FUNCTION_BLOCK Axis
//VAR_INPUT	
//END_VAR
VAR_OUTPUT
	Axis_Error			: BOOL;				// Error signal
	Axis_ErrorID		: UDINT;			// Error ID
	Axis_Moves			: BOOL;				// Status of moving
END_VAR
VAR
	// =============== Done signals MC Block =================
	JogDone			    : BOOL;					// Status of function block MC_Jog
	ResetDone		    : BOOL;					// Status of function block MC_Reset
	HaltDone		    : BOOL;					// Status of function block MC_Halt
	HomeDone		    : BOOL;					// Status of function block MC_Home
  MoveAbsoluteDone : BOOL;        // Status of function block MC_MoveAbsolute
  ExtSetPiontDone 	: BOOL;         		// Status of function block MC_ExtSetPointGenDisable

	// =============== Control variables ======================
	//Home_Back_Start	: BOOL;
	//Drive_Home		: BOOL;
	
	// =============== State variables ========================
	Power_StatusEnable	: BOOL;					// Enable feedback
	
	// =============== Velocity, override =====================
	Velocity_Jog		: LREAL;				// Jog velocity
	Velocity_Move		: LREAL;				// Target velocity
	Velocity_Home		: LREAL;				// Home1 velocity
  Velocity_Home2    : LREAL;        // Home1 velocity   
	Velocity_Absolute	: LREAL;				// MoveAbsolute velocity
	Velocity_Relative	: LREAL;				// MoveRelative velocity
	fOverride 			: LREAL := 100.0;		// Override 100%
	
	// =============== Trigger function blocks ================
	
	TriggerHalt	: R_TRIG;				// Trigger to recognize rising edge of halt input
	TriggerReset : R_TRIG;				// Trigger to recognize rising edge of reset input
	
	// =============== Axis reference =========================
	AxisRef			: AXIS_REF;				// Axis reference (process data plc/nc)
	
	// =============== About axis turque ====================
	Axis_Current_Turque 	: INT;
  	Axis_Max_Turque       	: INT;
	// ================= Sensor FeedBack ====================
  Proximity_Switch      : DINT;
  
	// =============== Motion function blocks =================
	Axis_Power 			: MC_Power;				// FB for enable and override			[上电]
	Axis_Home			: MC_Home;				// FB for axis home						[找零]
	Axis_Reset 			: MC_Reset;				// FB to reset axis						[复位]
	Axis_Jog			: MC_Jog;				// FB to jog axis						[点动]
	Axis_Stop 			: MC_Stop;				// FB to stop axis						[停止]
	Axis_Halt			: MC_Halt;				// FB to halt axis						[停止]
	Axis_Move			: MC_MoveVelocity;		// FB to move axis (velocity movement)	[匀速运动]
	Axis_MoveAbsolute 	: MC_MoveAbsolute;		// FB to move axis absolutely			[绝对位置运动]
	Axis_MoveRelative	: MC_MoveRelative;		// FB to move axis relatively			[相对位置运动]
  	Axis_ActPosition  : MC_ReadActualPosition; // FB to read the actual position of axis  [读取电机轴的实际位置]
	Axis_Delay			: Delay;				// FB to operate the delay program		[延迟程序]
	Axis_ExtSetPiontEnable	: MC_ExtSetPointGenEnable;	// FB to enable extsetpoint		[外部函数发生使能]
	Axis_ExtSetPiontDisable	: MC_ExtSetPointGenDisable;	// FB to disable extsetpoint	[外部函数结束使能]
  
  // =============== Timer =================
  Delay         : TON;          //[定时器]
END_VAR

PROPERTY ActPosition : LREAL
GET
Axis_ActPosition( Axis:= AxisRef, Enable:= TRUE );
ActPosition := Axis_ActPosition.Position;
END_GET
END_PROPERTY

PROPERTY Current_Turque_Value : INT
GET
Current_Turque_Value := Axis_Current_Turque;
END_GET
SET
Axis_Current_Turque := Current_Turque_Value;
END_SET
END_PROPERTY

METHOD ExtSetPoint
VAR_INPUT
	Drive_ExtSetPointEnable 	: BOOL;		// 使能外部信号开始信号
	Drive_ExtSetPointDisable 	: BOOL;		// 使能外部信号结束信号
	ExSetPosition				: LREAL;	// 外部信号位置
	//Axis_Current_Turque 		: INT;		// 边界条件：丝杠位置到达两端卡死
END_VAR
// =======================外部信号发生程序==========================

IF NOT Axis_ExtSetPiontEnable.Error THEN
	Axis_ExtSetPiontEnable(	Axis:= AxisRef, 
							Execute:= Drive_ExtSetPointEnable, 
							Position:= ExSetPosition, 
							PositionType:= POSITIONTYPE_ABSOLUTE );
END_IF

IF Axis_ExtSetPiontEnable.Done THEN
	ExtSetPiontDone := 1;
	MC_ExtSetPointGenFeed(	Position:= ExSetPosition, 
							Velocity:= 10, 
							Acceleration:= 10, 
							Direction:= 1, 		// 1 = positive direction
							Axis:= AxisRef );
END_IF	

IF NOT Axis_ExtSetPiontDisable.Error THEN 
	Axis_ExtSetPiontDisable(	Axis:= AxisRef, 
								Execute:= Drive_ExtSetPointDisable);
END_IF
								
IF Axis_ExtSetPiontEnable.Error OR Axis_ExtSetPiontDisable.Error OR ABS(Axis_Current_Turque) > Axis_Max_Turque THEN
	IF Axis_ExtSetPiontEnable.Error OR Axis_ExtSetPiontDisable.Error THEN
		Axis_Error		:= TRUE;
		Axis_ErrorID 	:= Axis_Home.ErrorID;
	END_IF
	Axis_ExtSetPiontEnable(	Axis:= AxisRef, 
							Execute:= 0 );
	Axis_ExtSetPiontDisable(	Axis:= AxisRef, 
								Execute:= 1);
END_IF
END_METHOD

METHOD Halt : BOOL
VAR_INPUT
	DriveHalt		: BOOL;					// Request stop
END_VAR
// =======================电机运动停止程序==========================

IF DriveHalt THEN
	// Move Execute FALSE
	Axis_Move(	Execute	:= FALSE,
				Axis 	:= AxisRef);
ELSE
	// Reset done signal
	HaltDone := FALSE;
END_IF

// Trigger
TriggerHalt(CLK := DriveHalt);

IF TriggerHalt.Q THEN
	Axis_Halt(	Execute	:= TRUE,
				Axis 	:= AxisRef);
ELSE
	Axis_Halt(Axis := AxisRef);
END_IF

// Done / Error / Command aborted
IF Axis_Halt.Done OR Axis_Halt.Error OR Axis_Halt.CommandAborted THEN
	Axis_Error		:= Axis_Halt.Error;
	Axis_ErrorID 	:= Axis_Halt.ErrorID;
	HaltDone 		:= Axis_Halt.Done;
	
	Axis_Move(	Execute	:= FALSE,
				Axis 	:= AxisRef);
				
	Axis_Halt(	Execute	:= FALSE,
				Axis 	:= AxisRef);
END_IF

// =========================================================
END_METHOD

METHOD Home
VAR_INPUT
	//Back_Start 				: BOOL;
	//Velocity_Home	:LREAL;
	//Axis_Current_Turque 	: INT;
	Drive_Home				: BOOL;
END_VAR

VAR
	HomeSet					: BOOL;
END_VAR
// =======================找零程序==========================
// 找零程序过程为：先让丝杠回退，到达机械限位后停止,并用程序将该位置置为零位

//======================丝杠回退========================
Jog_Backward(Drive_Jog_Backward:= Drive_Home);
Jog_Velocity := Velocity_Home;
	
IF NOT Axis_Home.Error THEN
	IF ABS(Axis_Current_Turque) > Axis_Max_Turque AND NOT HomeDone THEN
		Drive_Home :=0;
		Jog_Backward(Drive_Jog_Backward:= Drive_Home);
		Delay(IN:= NOT Delay.Q, PT:=T#200MS, Q=> , ET=> );
		Axis_Home( 	Axis:= AxisRef, 
					Execute:= Delay.Q, 
					Position:= 0, 
					HomingMode:= MC_Direct);
		HomeDone := Axis_Home.Done;
	END_IF
	IF HomeDone THEN
		Move_Absolute(Drive_Move_Absolute:= TRUE, Absolute_Position:= 10 );
		IF Axis_MoveAbsolute.Done THEN
			HomeDone := FALSE;
		END_IF
	END_IF
END_IF

(*IF HomeSet THEN
	Jog_Backward(Drive_Jog_Backward:= 0,  Axis_Current_Turque:= Axis_Current_Turque);
	HomeDone := 1;
END_IF*)

IF Axis_Home.Error OR Axis_Home.CommandAborted OR ABS(Axis_Current_Turque) < Axis_Max_Turque THEN
	IF Axis_Jog.Error THEN
		Axis_Error		:= TRUE;
		Axis_ErrorID 	:= Axis_Home.ErrorID;
	END_IF
	Axis_Home( 	Axis:= AxisRef, 
				Execute:= FALSE);
END_IF

// =========================================================
END_METHOD

PROPERTY Home_Velocity : LREAL
GET
Home_Velocity := Velocity_Home;
END_GET
SET
Velocity_Home := Home_Velocity;
END_SET
END_PROPERTY

METHOD Home2 : BOOL
VAR_INPUT
	Drive_Home		: BOOL;
END_VAR
// =======================找零程序==========================
// 找零程序过程为：先让丝杠回退，当传感器检测到金属表面并反馈信号后, 程序将该位置置为零位

//======================丝杠回退========================
Jog_Backward(Drive_Jog_Backward:= Drive_Home);
Jog_Velocity := Velocity_Home2;
	
IF NOT Axis_Home.Error THEN
	IF ABS(Proximity_Switch) = 64028672 AND NOT HomeDone THEN
		Drive_Home :=0;
		Jog_Backward(Drive_Jog_Backward:= Drive_Home);
		Delay(IN:= NOT Delay.Q, PT:=T#200MS, Q=> , ET=> );
		Axis_Home( 	Axis:= AxisRef, 
					Execute:= Delay.Q,
					Position:= 0, 
					HomingMode:= MC_Direct);
		HomeDone := Axis_Home.Done;
	END_IF
	IF HomeDone THEN
		Move_Absolute(Drive_Move_Absolute:= TRUE, Absolute_Position:= 20);
		IF Axis_MoveAbsolute.Done THEN
			HomeDone := FALSE;
		END_IF
	END_IF
END_IF

(*IF HomeSet THEN
	Jog_Backward(Drive_Jog_Backward:= 0,  Axis_Current_Turque:= Axis_Current_Turque);
	HomeDone := 1;
END_IF*)

IF Axis_Home.Error OR Axis_Home.CommandAborted OR ABS(Axis_Current_Turque) < Axis_Max_Turque THEN
	IF Axis_Jog.Error THEN
		Axis_Error		:= TRUE;
		Axis_ErrorID 	:= Axis_Home.ErrorID;
	END_IF
	Axis_Home( 	Axis:= AxisRef, 
				Execute:= FALSE);
END_IF

// =========================================================
END_METHOD

PROPERTY Home2_Velocity : LREAL
GET
Home2_Velocity := Velocity_Home2;
END_GET
SET
Velocity_Home2 := Home2_Velocity;
END_SET
END_PROPERTY

METHOD Jog_Backward
VAR_INPUT
	Drive_Jog_Backward	: BOOL;				//点动后退使能信号
	//Velocity_Jog		: LREAL;			//点动速度
	//Axis_Current_Turque : INT;				//边界条件：丝杠位置到达两端卡死
END_VAR
// =======================点动后退==========================
// 点动后退用在找零中的位置移动

IF NOT Axis_Jog.Error THEN
	Axis_Jog( 	Axis:= AxisRef, 
				JogForward:= 0, 
				JogBackwards:= Drive_Jog_Backward, 
				Mode:= MC_JOGMODE_CONTINOUS, 
				Velocity:= Velocity_Jog);
END_IF

IF Axis_Jog.Error OR Axis_Jog.CommandAborted OR ABS(Axis_Current_Turque) > Axis_Max_Turque THEN
	IF Axis_Jog.Error THEN
		Axis_Error		:= TRUE;
		Axis_ErrorID 	:= Axis_Jog.ErrorID;
	END_IF
	
	Axis_Jog(	JogForward:= 0, 
				JogBackwards:= 0, 
				Axis := AxisRef);
END_IF

(*IF ABS(Axis_Current_Turque) <1000 AND JogDone =1 THEN
	Axis_Jog(	JogForward:= 0, 
				JogBackwards:= 0, 
				Axis := AxisRef);
	JogDone :=0;
END_IF*)
				
// =========================================================
END_METHOD

METHOD Jog_Forward : BOOL
VAR_INPUT
	Drive_Jog_Forward	: BOOL;				//点动前进使能信号
	//Velocity_Jog		: LREAL;			//点动速度
	//Axis_Current_Turque : INT;				//边界条件：丝杠位置到达两端卡死
END_VAR
// =======================点动前进==========================


IF NOT Axis_Jog.Error THEN
	Axis_Jog( 	Axis:= AxisRef, 
				JogForward:= Drive_Jog_Forward, 
				JogBackwards:= 0, 
				Mode:= MC_JOGMODE_CONTINOUS, 
				Velocity:= Velocity_Jog);
END_IF

IF Axis_Jog.Error OR Axis_Jog.CommandAborted OR ABS(Axis_Current_Turque) > Axis_Max_Turque THEN
	IF Axis_Jog.Error THEN
		Axis_Error		:= TRUE;
		Axis_ErrorID 	:= Axis_Jog.ErrorID;
	END_IF
	
	Axis_Jog(	JogForward:= 0, 
				JogBackwards:= 0, 
				Axis := AxisRef);
END_IF

(*IF ABS(Axis_Current_Turque) <1000 AND JogDone =1 THEN
	Axis_Jog(	JogForward:= 0, 
				JogBackwards:= 0, 
				Axis := AxisRef);
	JogDone :=0;
END_IF*)
				
// =========================================================
END_METHOD

// =======================读写点动程序中的速度值==========================

PROPERTY Jog_Velocity : LREAL
GET
Jog_Velocity := Velocity_Jog;
END_GET
SET
Velocity_Jog := Jog_Velocity;
END_SET
END_PROPERTY

PROPERTY Max_Turque_Value : INT
SET
Axis_Max_Turque := Max_Turque_Value;
END_SET
END_PROPERTY

METHOD Move_Absolute
VAR_INPUT
	Drive_Move_Absolute : BOOL;				// 运动使能信号
	Absolute_Position	: LREAL;			// 绝对运动位置
	//Move_Velocity		: LREAL;			// 运动速度
	//Axis_Current_Turque : INT;			// 边界条件：丝杠位置到达两端卡死
END_VAR
// =======================绝对运动==========================

IF NOT Axis_MoveAbsolute.Error THEN
	Axis_MoveAbsolute(	Axis:= AxisRef, 
						Execute:= Drive_Move_Absolute, 
						Position:= Absolute_Position, 
						Velocity:= Velocity_Absolute, 
						BufferMode:= MC_Aborting );
	MoveAbsoluteDone := Axis_MoveAbsolute.Done;			// 运动到指定位置后置位
END_IF

IF Axis_MoveAbsolute.Error OR Axis_MoveAbsolute.CommandAborted OR ABS(Axis_Current_Turque) > Axis_Max_Turque THEN
	IF Axis_MoveAbsolute.Error THEN
		Axis_Error		:= TRUE;
		Axis_ErrorID 	:= Axis_MoveAbsolute.ErrorID;
	END_IF
	
	Axis_MoveAbsolute(	Axis:= AxisRef, 
						Execute:= 0, 
						BufferMode:= MC_Aborting);
END_IF

// =========================================================
END_METHOD

// =======================读写绝对运动程序中的速度值==========================

PROPERTY Move_Absolute_Velocity : LREAL
GET
Move_Absolute_Velocity := Velocity_Absolute;
END_GET
SET
Velocity_Absolute := Move_Absolute_Velocity;
END_SET
END_PROPERTY

METHOD Move_Backward
VAR_INPUT
	Move_Backward_Start : BOOL;					//匀速后退使能信号
	//Axis_Current_Turque : INT;					//边界条件：丝杠位置到达两端卡死
END_VAR
// =======================匀速后退==========================

// Not error
IF NOT Axis_Move.Error THEN
	Axis_Move(	Execute 	:= Move_Backward_Start,
				Velocity 	:= Velocity_Move,
				Direction 	:= MC_Negative_Direction,
				Axis 		:= AxisRef );
END_IF

// Error / Command aborted
IF Axis_Move.Error OR Axis_Move.CommandAborted OR ABS(Axis_Current_Turque) > Axis_Max_Turque THEN
	IF Axis_Move.Error THEN
		Axis_Error		:= TRUE;
		Axis_ErrorID 	:= Axis_Move.ErrorID;
	END_IF
	
	Axis_Move(	Execute	:= FALSE,
				Axis 	:= AxisRef);
END_IF

// =========================================================
END_METHOD

METHOD Move_Fordward
VAR_INPUT
	Move_Forward_Start : BOOL;					//匀速前进使能信号
	//Axis_Current_Turque : INT;					//边界条件：丝杠位置到达两端卡死
END_VAR
// =======================匀速前进==========================

// Not error
IF NOT Axis_Move.Error THEN
	Axis_Move(	Execute 	:= Move_Forward_Start,
				Velocity 	:= Velocity_Move,
				Direction 	:= MC_Positive_Direction,
				Axis 		:= AxisRef );
END_IF

// Error / Command aborted
IF Axis_Move.Error OR Axis_Move.CommandAborted OR ABS(Axis_Current_Turque) > Axis_Max_Turque THEN
	IF Axis_Move.Error THEN
		Axis_Error		:= TRUE;
		Axis_ErrorID 	:= Axis_Move.ErrorID;
	END_IF
	
	Axis_Move(	Execute	:= FALSE,
				Axis 	:= AxisRef);
END_IF

// =========================================================
END_METHOD

METHOD Move_Relative
VAR_INPUT
	Drive_Move_Relative		: BOOL;				// 运动使能信号
	Relative_Position		: LREAL;			// 相对运动位置
	//Move_Velocity			: LREAL;			// 运动速度
	//Axis_Current_Turque 	: INT;				// 边界条件：丝杠位置到达两端卡死
END_VAR
// =======================相对运动==========================

IF NOT Axis_MoveRelative.Error THEN
	Axis_MoveRelative(	Axis:= AxisRef, 
						Execute:= Drive_Move_Relative, 
						Distance:= Relative_Position, 
						Velocity:= Velocity_Relative, 
						BufferMode:= MC_Aborting );
END_IF

IF Axis_MoveRelative.Error OR Axis_MoveRelative.CommandAborted OR ABS(Axis_Current_Turque) > Axis_Max_Turque THEN
	IF Axis_MoveRelative.Error THEN
		Axis_Error		:= TRUE;
		Axis_ErrorID 	:= Axis_MoveRelative.ErrorID;
	END_IF
	
	Axis_MoveRelative(	Axis:= AxisRef, 
						Execute:= 0, 
						BufferMode:= MC_Aborting);
END_IF

// =========================================================
END_METHOD

// =======================读写相对运动程序中的速度值==========================

PROPERTY Move_Relative_Velocity : LREAL
GET
Move_Relative_Velocity := Velocity_Relative;
END_GET
SET
Velocity_Relative := Move_Relative_Velocity;
END_SET
END_PROPERTY

PROPERTY Move_Velocity : LREAL
GET
Move_Velocity := Velocity_Move;
END_GET
SET
Velocity_Move :=Move_Velocity :=10;
END_SET
END_PROPERTY

METHOD Power
VAR_INPUT
	Axis_Enable : BOOL;
END_VAR
// =======================上电程序==========================

Axis_Power(	Enable 			:= Axis_Enable, 
			Enable_Positive	:= Axis_Enable, 
			Enable_Negative	:= Axis_Enable, 
			Override		:= fOverride,
			Axis			:= AxisRef,
			Status			=> Power_StatusEnable);
			
IF Axis_Power.Error THEN
	Axis_Error		:= TRUE;
	Axis_ErrorID 	:= Axis_Power.ErrorID;
END_IF

AxisRef.ReadStatus();

Axis_Moves := AxisRef.Status.Moving;

// ==========================================================
END_METHOD

PROPERTY Proximity_Switch_FeedBack : DINT
SET
Proximity_Switch := Proximity_Switch_FeedBack;
END_SET
END_PROPERTY

METHOD Reset
VAR_INPUT
	Drive_Reset		: BOOL;					// Request reset
END_VAR
// =====================驱动重置程序==========================

IF NOT Drive_Reset THEN
	ResetDone 	:= FALSE;
END_IF

// Trigger(触发器)
TriggerReset(CLK := Drive_Reset);

IF TriggerReset.Q THEN
	HaltDone 	:= FALSE;
	
	Axis_Reset(Execute := TRUE, Axis := AxisRef);
ELSE
	Axis_Reset(Axis := AxisRef);
END_IF

// Done / Error
IF Axis_Reset.Done OR Axis_Reset.Error THEN
	Axis_Error		:= Axis_Reset.Error;
	Axis_ErrorID 	:= Axis_Reset.ErrorID;
	ResetDone 		:= Axis_Reset.Done;

	Axis_Reset(	Execute	:= FALSE, Axis 	:= AxisRef);
END_IF

// =========================================================
END_METHOD

PROPERTY State_ExtSetPiontDone : BOOL
GET
State_ExtSetPiontDone := ExtSetPiontDone;
END_GET
END_PROPERTY

// =======================回零结束信号==========================

PROPERTY State_HomeDone : BOOL
GET
State_HomeDone := HomeDone;
END_GET
END_PROPERTY

// =======================点动结束信号==========================

PROPERTY State_JogDone : BOOL
GET
State_JogDone := JogDone;
END_GET
END_PROPERTY

PROPERTY State_MoveAbsoluteDone : BOOL
GET
State_MoveAbsoluteDone := MoveAbsoluteDone;
END_GET
END_PROPERTY

// =======================上电状态信号==========================

PROPERTY State_PowerStatus : BOOL
GET
State_PowerStatus := Power_StatusEnable;
END_GET
END_PROPERTY

// =======================复位结束信号==========================

PROPERTY State_ResetDone : BOOL
GET
State_ResetDone := ResetDone;
END_GET
END_PROPERTY

END_FUNCTION_BLOCK

(* stored: Version 1.1.0.1, ProductVersion 3.1.4020.12
   POU Axis: Id {752ec826-01be-4872-838e-fdec6a999a4b}, SpecialFunc None
   Property ActPosition: Id {3015e613-88a6-44b7-bfd3-2c06df6f075d}
   Get Get: Id {a1550c61-e344-45b9-84a9-b4c92d3e44f5}
   Property Current_Turque_Value: Id {3a2f771d-3376-4640-bd97-650af6e34455}
   Get Get: Id {cf61b5f8-2ee8-4892-af0b-6df01ee01050}
   Set Set: Id {454d6b57-9848-48a1-bdc6-2e4c4bcfbc97}
   Method ExtSetPoint: Id {e3dd3d6b-d150-49a2-a8d7-a7990a606e4c}
   Method Halt: Id {d7ff254f-2dd7-462f-bdbd-9197c2ffdaa3}
   Method Home: Id {313e1eef-e597-492a-a006-a8453e584cfd}
   Property Home_Velocity: Id {075d0823-6614-4698-9d00-5a9266b58e8c}
   Get Get: Id {337c8281-9e84-4066-80f8-1804a324ddb1}
   Set Set: Id {28f71fe8-0908-4a45-b6fa-862d0622a7a8}
   Method Home2: Id {538e8ca7-d46b-41f9-930c-142666bfb84c}
   Property Home2_Velocity: Id {29542bf1-ba67-49a9-803d-762403c92f58}
   Get Get: Id {fe78f786-10a8-4f98-9e65-95fb7c4427c2}
   Set Set: Id {7e1f886e-1b8d-4d9a-9fc1-c6d7443f0295}
   Method Jog_Backward: Id {99d13956-4937-48a4-92d1-297e5120f462}
   Method Jog_Forward: Id {9deceb4f-22e3-43d3-abba-cc65da0a988f}
   Property Jog_Velocity: Id {fbf70f23-ccbc-42f7-9290-364343308531}
   Get Get: Id {777f885d-c13b-46bb-a81c-11c9d0c034b5}
   Set Set: Id {3493f918-b8b5-4bfd-88eb-49ef90625a72}
   Property Max_Turque_Value: Id {c8624b49-e9f6-4c92-b644-367354523826}
   Set Set: Id {d52428b7-2c03-4786-a6ff-9fe9a6b65b24}
   Method Move_Absolute: Id {90058d1c-d052-4ccf-9289-5faf8ddb84ca}
   Property Move_Absolute_Velocity: Id {7cb9ac45-b7a3-4012-b6de-6d6ce49b5a54}
   Get Get: Id {69b3b0a0-70e4-4a5d-b413-ab7229a2e9bd}
   Set Set: Id {226c6ce0-f119-45e3-aed2-044f6ed96e56}
   Method Move_Backward: Id {d07db03f-d706-432b-92a0-251009b4d606}
   Method Move_Fordward: Id {30d70636-f830-44c4-adf2-54f90ee067a6}
   Method Move_Relative: Id {7b541efd-c3a2-463f-9025-d3f3cd116050}
   Property Move_Relative_Velocity: Id {10d568b7-1224-4f3c-82dc-f2b473343afd}
   Get Get: Id {348afd78-8fc2-4019-a44e-c1c1383e294e}
   Set Set: Id {5825f81f-4221-4e2d-a800-e81839a342ef}
   Property Move_Velocity: Id {21dc1ad2-a805-4cc5-ba52-5eb4a3378ad2}
   Get Get: Id {1866d0e7-3c70-4d48-8eca-a37834a3ae08}
   Set Set: Id {22390785-422b-4fe3-a5a7-2a060fc5e62a}
   Method Power: Id {cc0985ad-b04b-4e99-b924-c7a9a3e5739c}
   Property Proximity_Switch_FeedBack: Id {266d5a90-626e-4237-baca-31f21f0c8e8c}
   Set Set: Id {4caf84bf-6035-4fe8-8acd-b0890ff2a20e}
   Method Reset: Id {dedc8057-c4ab-4248-b14b-274fa3c9288f}
   Property State_ExtSetPiontDone: Id {6243132d-fdac-4a44-aabc-1626db2c504e}
   Get Get: Id {707129e4-107c-4490-bb7b-c4d081868570}
   Property State_HomeDone: Id {b05cc381-4a45-4536-92f9-829385d416fe}
   Get Get: Id {264bc084-d205-492c-afbe-d826e47ed36b}
   Property State_JogDone: Id {3c0f115e-f80a-44b9-a70e-39bb83e64c81}
   Get Get: Id {0fe6b904-9b2c-4f79-ad95-929babff25cb}
   Property State_MoveAbsoluteDone: Id {7b7a8b76-a437-47fb-99a9-6a9d632d1395}
   Get Get: Id {c74d3577-a7ec-4111-94f6-46d87e085a5c}
   Property State_PowerStatus: Id {26f2d544-ee3f-4b26-afb9-71118906e7d1}
   Get Get: Id {f32eea30-ecfd-40aa-98ad-396678666aa2}
   Property State_ResetDone: Id {e8bc9f4f-5bd7-4f76-a8c5-8b726ec5b1c8}
   Get Get: Id {305c7aa0-f515-4867-a0e8-4b3fd35a9f3f} *)
